FUNCTION_BLOCK WaterSensor
  (* Standard: 61499-2 *)
  (* Version 0.2, 2003-12-04, JHC, Rockwell Automation, Renamed for better indexing. *)
  (* Version 0.1, 2002-11-05, JHC, Rockwell Automation, Corrected missing ST element in Algorithm REQ. *)
  (* Version 0.0, 2000-05-30, JHC, Rockwell Automation *)
  (* Compiler header: package fb.rt.benchmarks.watermonitor; *)
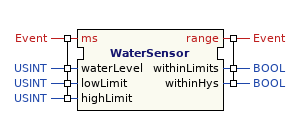
  EVENT_INPUT
    ms WITH waterLevel, lowLimit, highLimit; (* millisecond *)
  END_EVENT
  EVENT_OUTPUT
    range WITH withinLimits, withinHys;
  END_EVENT
  VAR_INPUT
    waterLevel : USINT := 150;
    lowLimit : USINT := 100;
    highLimit : USINT := 200;
  END_VAR
  VAR_OUTPUT
    withinLimits : BOOL := true;
    withinHys : BOOL := true;
  END_VAR
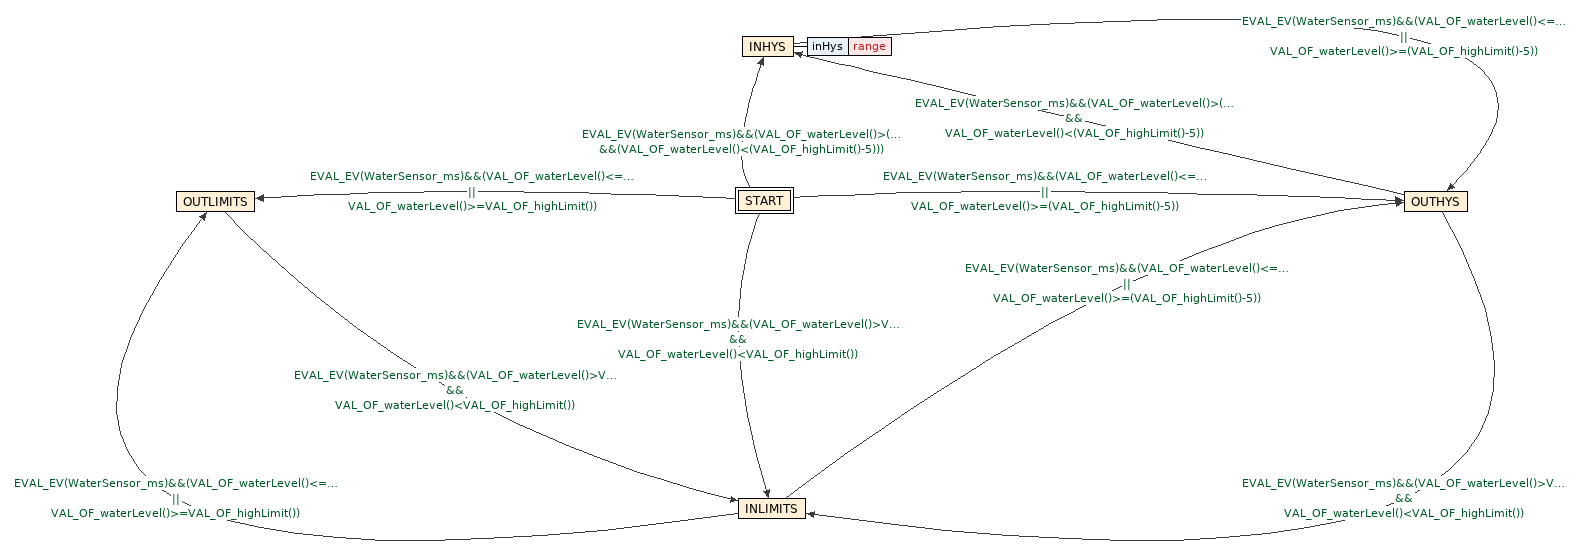
  EC_STATES
    START; (* Initial State *)
    INHYS : inHys -> range; (* in hysterisis *)
    INLIMITS; (* within limts *)
    OUTLIMITS; (* outside limits *)
    OUTHYS; (* outside hysterisis *)
  END_STATES
  EC_TRANSITIONS
    START TO INHYS := EVAL_EV(WaterSensor_ms)&&(VAL_OF_waterLevel()>(VAL_OF_lowLimit()+5)  &&(VAL_OF_waterLevel()<(VAL_OF_highLimit()-5)));
    START TO OUTHYS := EVAL_EV(WaterSensor_ms)&&(VAL_OF_waterLevel()<=(VAL_OF_lowLimit()+5) || VAL_OF_waterLevel()>=(VAL_OF_highLimit()-5));
    START TO INLIMITS := EVAL_EV(WaterSensor_ms)&&(VAL_OF_waterLevel()>VAL_OF_lowLimit() && VAL_OF_waterLevel()<VAL_OF_highLimit());
    START TO OUTLIMITS := EVAL_EV(WaterSensor_ms)&&(VAL_OF_waterLevel()<=VAL_OF_lowLimit() || VAL_OF_waterLevel()>=VAL_OF_highLimit());
    INHYS TO OUTHYS := EVAL_EV(WaterSensor_ms)&&(VAL_OF_waterLevel()<=(VAL_OF_lowLimit()+5) || VAL_OF_waterLevel()>=(VAL_OF_highLimit()-5));
    OUTHYS TO INHYS := EVAL_EV(WaterSensor_ms)&&(VAL_OF_waterLevel()>(VAL_OF_lowLimit()+5) && VAL_OF_waterLevel()<(VAL_OF_highLimit()-5));
    OUTHYS TO INLIMITS := EVAL_EV(WaterSensor_ms)&&(VAL_OF_waterLevel()>VAL_OF_lowLimit() && VAL_OF_waterLevel()<VAL_OF_highLimit());
    INLIMITS TO OUTHYS := EVAL_EV(WaterSensor_ms)&&(VAL_OF_waterLevel()<=(VAL_OF_lowLimit()+5) || VAL_OF_waterLevel()>=(VAL_OF_highLimit()-5));
    INLIMITS TO OUTLIMITS := EVAL_EV(WaterSensor_ms)&&(VAL_OF_waterLevel()<=VAL_OF_lowLimit() || VAL_OF_waterLevel()>=VAL_OF_highLimit());
    OUTLIMITS TO INLIMITS := EVAL_EV(WaterSensor_ms)&&(VAL_OF_waterLevel()>VAL_OF_lowLimit() && VAL_OF_waterLevel()<VAL_OF_highLimit());
  END_TRANSITIONS
  ALGORITHM inHys IN ST: (* Normally executed algorithm *)
VAL_OF_withinHys()= 1;
VAL_OF_withinLimits ()= 1;
  END_ALGORITHM
  ALGORITHM outHys IN ST:
VAL_OF_withinHys()= 0;
  END_ALGORITHM
  ALGORITHM inLimits IN ST: (* Initialization algorithm *)
VAL_OF_withinLimits ()= 1;
  END_ALGORITHM
  ALGORITHM outLimits IN ST:
VAL_OF_withinLimits ()= 0;
VAL_OF_withinHys()= 0;
  END_ALGORITHM
END_FUNCTION_BLOCK
